PROGRAM PRG_MachineSafety
VAR
	bFirstCycle 	: BOOL := TRUE;
	fbMachineSafety : FB_MachineSafety;
END_VAR

(* First cycle of visu controler run*)
IF bFirstCycle THEN
	bFirstCycle := FALSE;
	
	(* Assign machine controler reference to Shell API*)
	stShell.stPlatform.ref_MachineSafety REF= fbMachineSafety;
	
END_IF

(* Cyclic run of machine safety *)
fbMachineSafety();

END_PROGRAM

(* stored: Version 1.1.0.1, ProductVersion 3.1.4024.9
   POU PRG_MachineSafety: Id {537b7dc6-6c67-40ee-bee2-17822a50d8a9}, SpecialFunc None *)
